// TIA Portal V18 export
FUNCTION_BLOCK "ST10_Flow24_LUnloadingTrans"   // FB1094, GRAPH
VERSION : 0.1
// stored: AcknowledgeErrorsRequired false, AutoNumber false, GraphVersion 6.0, InitialValuesAcquisition false, IsIECCheckEnabled false, LanguageInNetworks LAD, LockOperatingMode false, PermanentILProcessingInMANMode false, SetENOAutomatically false, SkipSteps false, UDAEnableTagReadback false, WithAlarmHandling true
   // inherited from GRAPH_BASE
   VAR
      OFF_SQ_BASE : Bool;
   END_VAR
   VAR_INPUT
      iSysInface : "RCS_SysComInterface_V1";
   END_VAR
   VAR_IN_OUT
      ioPM_Inface : "RCS_PMInterface_V1";
      ioStatus : Int;
   END_VAR
   VAR
      sCtrlMode { S7_SetPoint := 'True'} : "SysFlowCtrlGraph";
      sUpdMES_Data : Bool;   // 更新MES数据
      工件放行中 : Bool;
      前站站号 { ExternalAccessible := 'False'; ExternalVisible := 'False'; ExternalWritable := 'False'} : UInt;
      本站站号 { ExternalAccessible := 'False'; ExternalVisible := 'False'; ExternalWritable := 'False'} : UInt;
      弹窗Temp : Array[1..10] of Int;
      AlarmID : Int;
      TON { S7_SetPoint := 'True'} : Array[0..10] of TON_TIME;
      TOF { S7_SetPoint := 'True'} : Array[0..10] of TOF_TIME;
      sUP { S7_SetPoint := 'True'} : Array[0..10] of Bool;
      更新RFID完成 : Bool;
   END_VAR
   VAR_TEMP
      Tempresult : USInt;
      本站站号乘10 : UInt;
   END_VAR
   // // TON[0] : 托盘流入1托盘到位传感器 / iA-Rotating product Check
   // // TON[1] : 托盘流入1托盘到位传感器
   // // TON[2] : 托盘流入1产品有无传感器
   // // TON[3] : 托盘流入1产品有无传感器
   // // TON[4] : 托盘流入1姿态检测光电2
   // // TON[5] : 托盘流入1姿态检测光电3
   // // TON[0].Q : 托盘流入1托盘到位 / iA-Rotating product Check
   // // TON[1].Q : 托盘流入1托盘无
   // // TON[2].Q : 托盘流入1有产品
   // // TON[3].Q : 托盘流入1无产品
   // // TON[4].Q : 托盘流入1姿态检测光电2
   // // TON[5].Q : 托盘流入1姿态检测光电3
   // // TOF[1] : iA-Rotating product Check
BEGIN
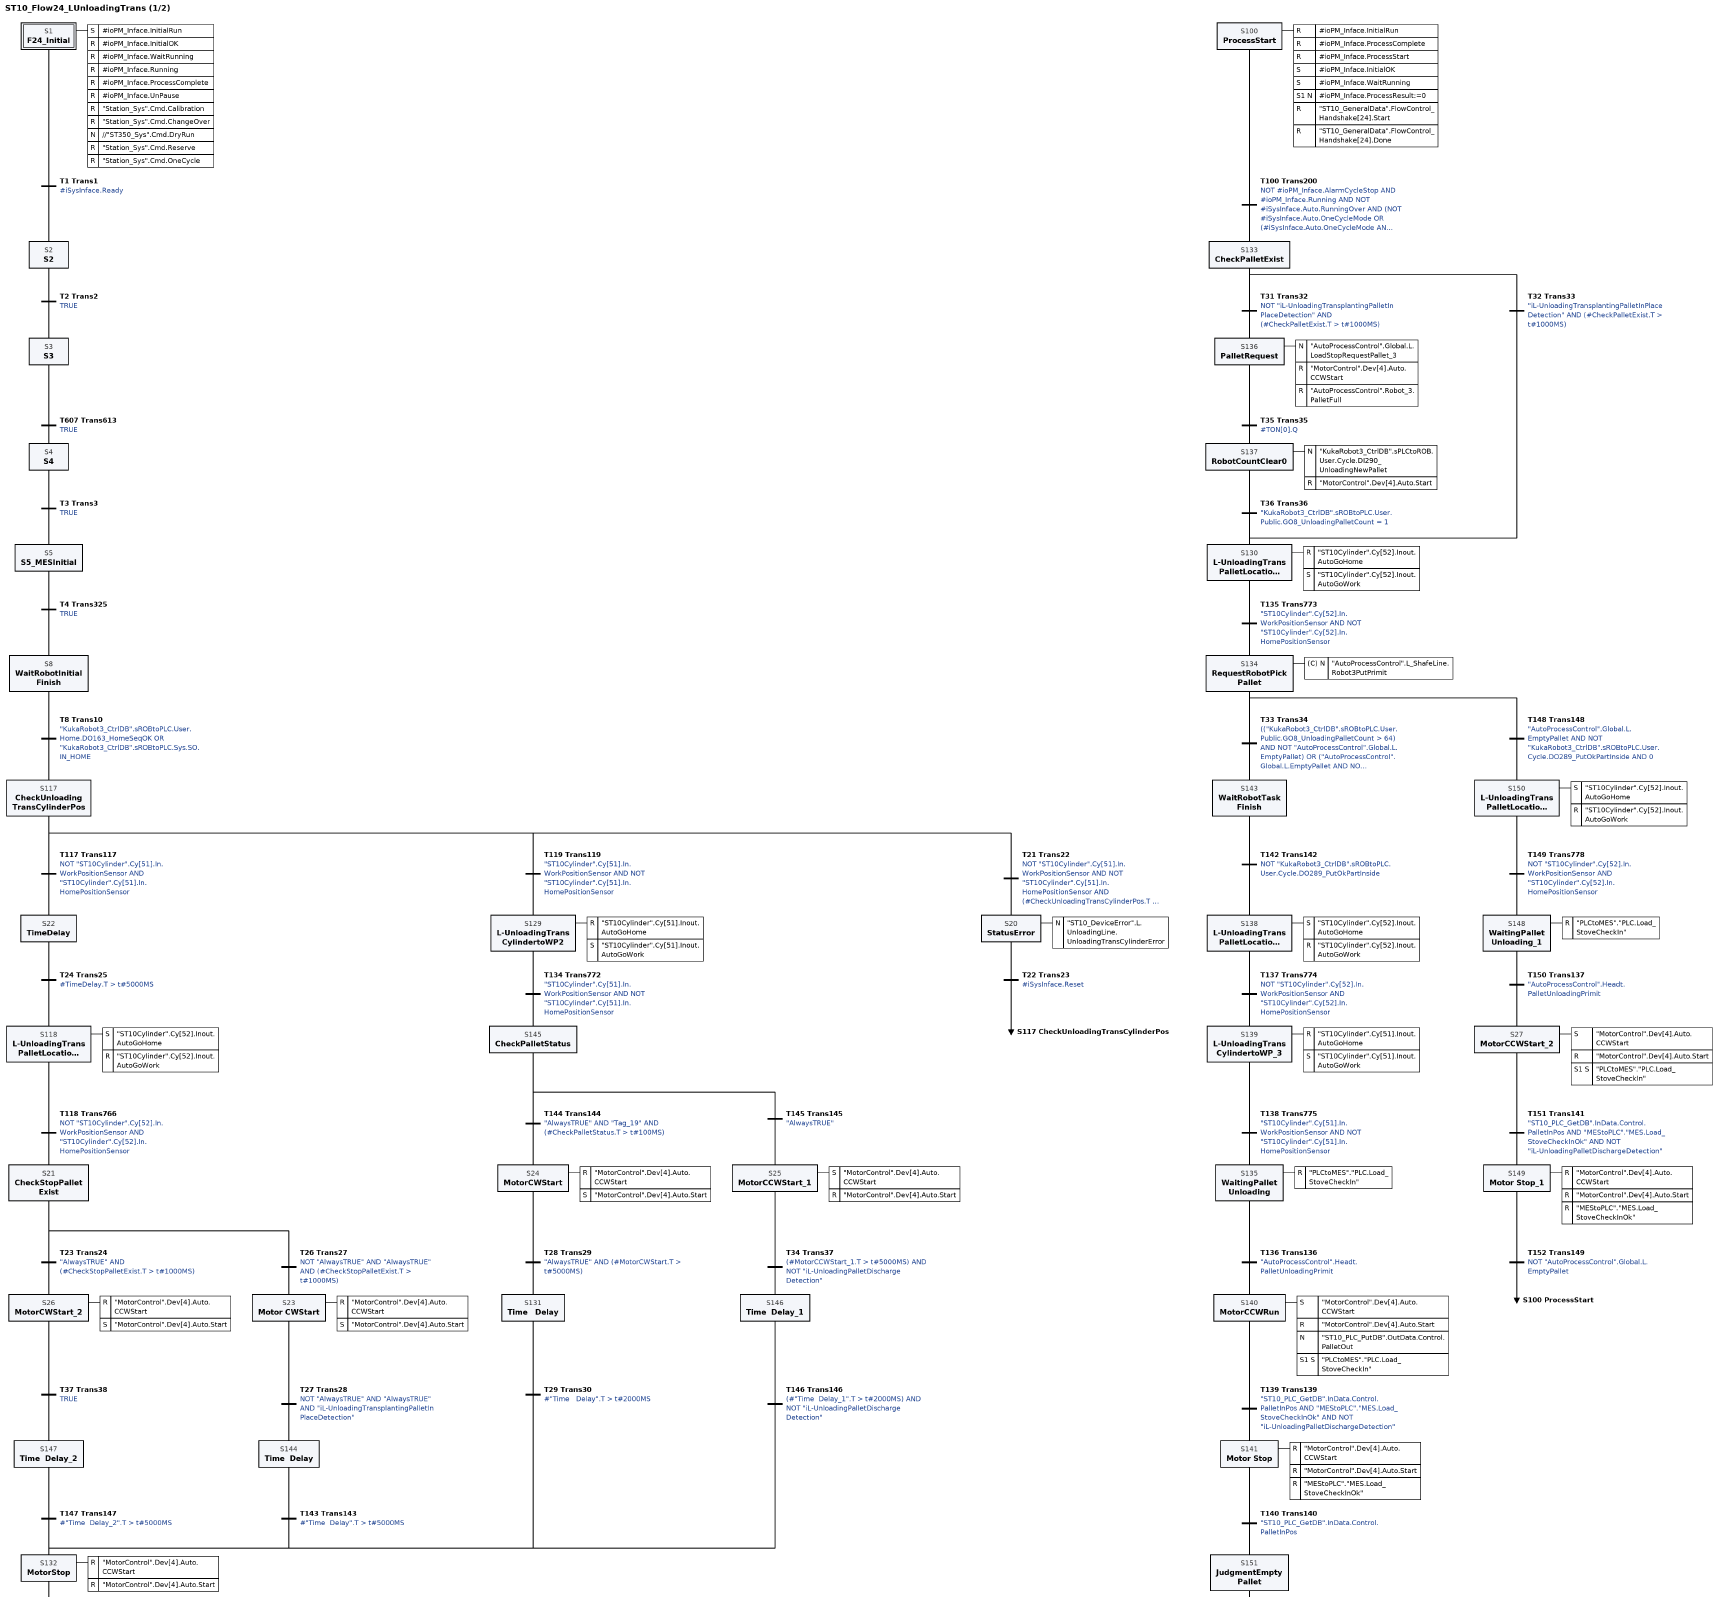
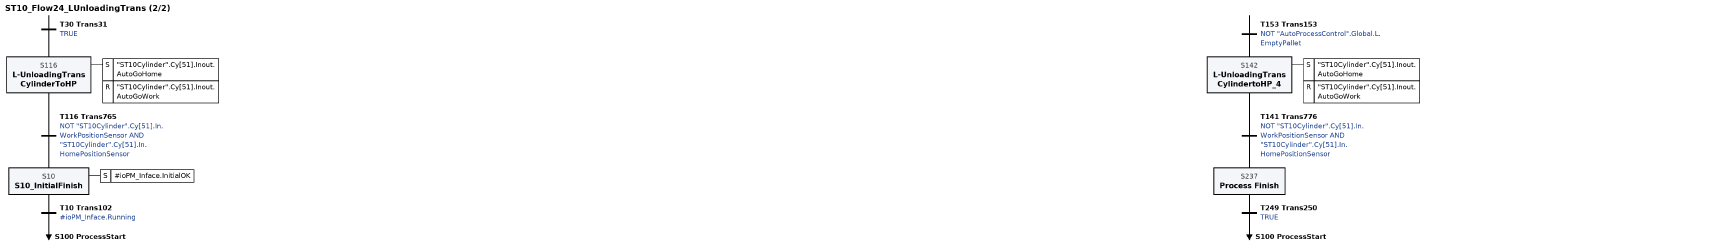
   // permanent pre-instructions
   NETWORK 1
      #TON[10].TON(IN := "AlwaysTRUE" AND "Station_Sys".Alarm.ImmediatelyStop, PT := T#300ms);
      #ioPM_Inface.AlarmImdilyStop := #TON[10].Q;
      #ioPM_Inface.AlarmCycleStop := "AlwaysTRUE" AND "Station_Sys".Alarm.CycleStop;
   NETWORK 2
      IF NOT False THEN
          #sCtrlMode(iSysInface := #iSysInface, ioPM_Inface := #ioPM_Inface, ioGraphCtrl := #RT_DATA.MOP);   // "SysFlowCtrlGraph"
      END_IF;
   NETWORK 3
      #TON[0].TON(IN := "AlwaysTRUE" AND "iL-UnloadingTransplantingPalletInPlaceDetection", PT := t#1000ms);   // 工位11有托盘
      #TOF[1].TOF(IN := "AlwaysTRUE" AND NOT "iL-UnloadingTransplantingPalletInPlaceDetection", PT := T#300ms);   // 工位无托盘
      #TON[2].TON(IN := "AlwaysTRUE", PT := T#300ms);
      #TOF[3].TOF(IN := "AlwaysTRUE", PT := T#300ms);
      #TON[4].TON(IN := "AlwaysTRUE", PT := T#300ms);
      #TOF[5].TOF(IN := "AlwaysTRUE", PT := T#300ms);
   NETWORK 4
      #前站站号 := 345;
      #本站站号 := 350;
   NETWORK 5
      IF "AlwaysTRUE" AND "MEStoPLC"."MES.Load_StoveCheckInOk" THEN
          "PLCtoMES"."PLC.Load_StoveCheckIn" := FALSE;
      END_IF;

   // sequencer 1: S01-S99 初始化 / S01-S99 Initial
   INITIAL_STEP F24_Initial:   // S1, max time T#10S, warning time T#7S
              S    #ioPM_Inface.InitialRun
              R    #ioPM_Inface.InitialOK
              R    #ioPM_Inface.WaitRunning
              R    #ioPM_Inface.Running
              R    #ioPM_Inface.ProcessComplete
              R    #ioPM_Inface.UnPause
              R    "Station_Sys".Cmd.Calibration
              R    "Station_Sys".Cmd.ChangeOver
                   //"ST350_Sys".Cmd.DryRun
              R    "Station_Sys".Cmd.Reserve
              R    "Station_Sys".Cmd.OneCycle
   END_STEP
   TRANSITION Trans1 FROM F24_Initial TO S2   // T1
      := #iSysInface.Ready;
   END_TRANSITION
   STEP S2:   // S2, max time T#10S, warning time T#7S
   END_STEP
   TRANSITION Trans2 FROM S2 TO S3   // T2
      := TRUE;
   END_TRANSITION
   STEP S4:   // S4, max time T#10S, warning time T#7S
   END_STEP
   TRANSITION Trans3 FROM S4 TO S5_MESInitial   // T3
      := TRUE;
   END_TRANSITION
   STEP S5_MESInitial:   // S5, max time T#10S, warning time T#7S
   END_STEP
   TRANSITION Trans325 FROM S5_MESInitial TO WaitRobotInitialFinish   // T4
      := TRUE;
   END_TRANSITION
   STEP S10_InitialFinish:   // S10, max time T#10S, warning time T#7S
              S    #ioPM_Inface.InitialOK
   END_STEP
   TRANSITION Trans102 FROM S10_InitialFinish TO ProcessStart   // T10, jump
      := #ioPM_Inface.Running;
   END_TRANSITION
   STEP S3:   // S3, max time T#10S, warning time T#7S
   END_STEP
   TRANSITION Trans613 FROM S3 TO S4   // T607
      := TRUE;
   END_TRANSITION
   STEP WaitRobotInitialFinish:   // S8, max time T#10S, warning time T#7S
   END_STEP
   TRANSITION Trans10 FROM WaitRobotInitialFinish TO CheckUnloadingTransCylinderPos   // T8
      := "KukaRobot3_CtrlDB".sROBtoPLC.User.Home.DO163_HomeSeqOK OR "KukaRobot3_CtrlDB".sROBtoPLC.Sys.SO.IN_HOME;
   END_TRANSITION
   STEP "Time   Delay":   // S131, max time T#10S, warning time T#7S
   END_STEP
   TRANSITION Trans30 FROM "Time   Delay" TO MotorStop   // T29
      := #"Time   Delay".T > t#2000MS;
   END_TRANSITION
   STEP CheckUnloadingTransCylinderPos:   // S117, max time T#10S, warning time T#7S
   END_STEP
   TRANSITION Trans117 FROM CheckUnloadingTransCylinderPos TO TimeDelay   // T117
      := NOT "ST10Cylinder".Cy[51].In.WorkPositionSensor AND "ST10Cylinder".Cy[51].In.HomePositionSensor;
   END_TRANSITION
   TRANSITION Trans119 FROM CheckUnloadingTransCylinderPos TO "L-UnloadingTransCylindertoWP2"   // T119
      := "ST10Cylinder".Cy[51].In.WorkPositionSensor AND NOT "ST10Cylinder".Cy[51].In.HomePositionSensor;
   END_TRANSITION
   TRANSITION Trans22 FROM CheckUnloadingTransCylinderPos TO StatusError   // T21
      := NOT "ST10Cylinder".Cy[51].In.WorkPositionSensor AND NOT "ST10Cylinder".Cy[51].In.HomePositionSensor AND (#CheckUnloadingTransCylinderPos.T > t#2000MS);
   END_TRANSITION
   STEP "L-UnloadingTransCylinderToHP":   // S116, max time T#10S, warning time T#7S
              S    "ST10Cylinder".Cy[51].Inout.AutoGoHome
              R    "ST10Cylinder".Cy[51].Inout.AutoGoWork
   END_STEP
   TRANSITION Trans765 FROM "L-UnloadingTransCylinderToHP" TO S10_InitialFinish   // T116
      := NOT "ST10Cylinder".Cy[51].In.WorkPositionSensor AND "ST10Cylinder".Cy[51].In.HomePositionSensor;
   END_TRANSITION
   STEP StatusError:   // S20, max time T#10S, warning time T#7S
              N    "ST10_DeviceError".L.UnloadingLine.UnloadingTransCylinderError
   END_STEP
   TRANSITION Trans23 FROM StatusError TO CheckUnloadingTransCylinderPos   // T22, jump
      := #iSysInface.Reset;
   END_TRANSITION
   STEP CheckStopPalletExist:   // S21, max time T#10S, warning time T#7S
   END_STEP
   TRANSITION Trans24 FROM CheckStopPalletExist TO MotorCWStart_2   // T23
      := "AlwaysTRUE" AND (#CheckStopPalletExist.T > t#1000MS);
   END_TRANSITION
   TRANSITION Trans27 FROM CheckStopPalletExist TO "Motor CWStart"   // T26
      := NOT "AlwaysTRUE" AND "AlwaysTRUE" AND (#CheckStopPalletExist.T > t#1000MS);
   END_TRANSITION
   STEP TimeDelay:   // S22, max time T#10S, warning time T#7S
   END_STEP
   TRANSITION Trans25 FROM TimeDelay TO "L-UnloadingTransPalletLocationCylinderHP_2"   // T24
      := #TimeDelay.T > t#5000MS;
   END_TRANSITION
   STEP "Motor CWStart":   // S23, max time T#10S, warning time T#7S
              R    "MotorControl".Dev[4].Auto.CCWStart
              S    "MotorControl".Dev[4].Auto.Start
   END_STEP
   TRANSITION Trans28 FROM "Motor CWStart" TO "Time  Delay"   // T27
      := NOT "AlwaysTRUE" AND "AlwaysTRUE" AND "iL-UnloadingTransplantingPalletInPlaceDetection";
   END_TRANSITION
   STEP MotorCWStart:   // S24, max time T#10S, warning time T#7S
              R    "MotorControl".Dev[4].Auto.CCWStart
              S    "MotorControl".Dev[4].Auto.Start
   END_STEP
   TRANSITION Trans29 FROM MotorCWStart TO "Time   Delay"   // T28
      := "AlwaysTRUE" AND (#MotorCWStart.T > t#5000MS);
   END_TRANSITION
   STEP "L-UnloadingTransCylindertoWP2":   // S129, max time T#10S, warning time T#7S
              R    "ST10Cylinder".Cy[51].Inout.AutoGoHome
              S    "ST10Cylinder".Cy[51].Inout.AutoGoWork
   END_STEP
   TRANSITION Trans772 FROM "L-UnloadingTransCylindertoWP2" TO CheckPalletStatus   // T134
      := "ST10Cylinder".Cy[51].In.WorkPositionSensor AND NOT "ST10Cylinder".Cy[51].In.HomePositionSensor;
   END_TRANSITION
   STEP MotorStop:   // S132, max time T#10S, warning time T#7S
              R    "MotorControl".Dev[4].Auto.CCWStart
              R    "MotorControl".Dev[4].Auto.Start
   END_STEP
   TRANSITION Trans31 FROM MotorStop TO "L-UnloadingTransCylinderToHP"   // T30
      := TRUE;
   END_TRANSITION
   STEP "L-UnloadingTransPalletLocationCylinderHP_2":   // S118, max time T#10S, warning time T#7S
              S    "ST10Cylinder".Cy[52].Inout.AutoGoHome
              R    "ST10Cylinder".Cy[52].Inout.AutoGoWork
   END_STEP
   TRANSITION Trans766 FROM "L-UnloadingTransPalletLocationCylinderHP_2" TO CheckStopPalletExist   // T118
      := NOT "ST10Cylinder".Cy[52].In.WorkPositionSensor AND "ST10Cylinder".Cy[52].In.HomePositionSensor;
   END_TRANSITION
   STEP "Time  Delay":   // S144, max time T#10S, warning time T#7S
   END_STEP
   TRANSITION Trans143 FROM "Time  Delay" TO MotorStop   // T143
      := #"Time  Delay".T > t#5000MS;
   END_TRANSITION
   STEP CheckPalletStatus:   // S145, max time T#10S, warning time T#7S
   END_STEP
   TRANSITION Trans144 FROM CheckPalletStatus TO MotorCWStart   // T144
      := "AlwaysTRUE" AND "Tag_19" AND (#CheckPalletStatus.T > t#100MS);
   END_TRANSITION
   TRANSITION Trans145 FROM CheckPalletStatus TO MotorCCWStart_1   // T145
      := "AlwaysTRUE";
   END_TRANSITION
   STEP MotorCCWStart_1:   // S25, max time T#10S, warning time T#7S
              S    "MotorControl".Dev[4].Auto.CCWStart
              R    "MotorControl".Dev[4].Auto.Start
   END_STEP
   TRANSITION Trans37 FROM MotorCCWStart_1 TO "Time  Delay_1"   // T34
      := (#MotorCCWStart_1.T > t#5000MS) AND NOT "iL-UnloadingPalletDischargeDetection";
   END_TRANSITION
   STEP "Time  Delay_1":   // S146, max time T#10S, warning time T#7S
   END_STEP
   TRANSITION Trans146 FROM "Time  Delay_1" TO MotorStop   // T146
      := (#"Time  Delay_1".T > t#2000MS) AND NOT "iL-UnloadingPalletDischargeDetection";
   END_TRANSITION
   STEP MotorCWStart_2:   // S26, max time T#10S, warning time T#7S
              R    "MotorControl".Dev[4].Auto.CCWStart
              S    "MotorControl".Dev[4].Auto.Start
   END_STEP
   TRANSITION Trans38 FROM MotorCWStart_2 TO "Time  Delay_2"   // T37
      := TRUE;
   END_TRANSITION
   STEP "Time  Delay_2":   // S147, max time T#10S, warning time T#7S
   END_STEP
   TRANSITION Trans147 FROM "Time  Delay_2" TO MotorStop   // T147
      := #"Time  Delay_2".T > t#5000MS;
   END_TRANSITION

   // sequencer 2: S100-S199 等待到位 / S100-S199 CheckPalletStatus
   STEP ProcessStart:   // S100, max time T#10S, warning time T#7S
      // 自动等待开始运行
              R    #ioPM_Inface.InitialRun
              R    #ioPM_Inface.ProcessComplete
              R    #ioPM_Inface.ProcessStart
              S    #ioPM_Inface.InitialOK
              S    #ioPM_Inface.WaitRunning
          S1  N    #ioPM_Inface.ProcessResult:=0
              R    "ST10_GeneralData".FlowControl_Handshake[24].Start
              R    "ST10_GeneralData".FlowControl_Handshake[24].Done
   END_STEP
   TRANSITION Trans200 FROM ProcessStart TO CheckPalletExist   // T100
      := NOT #ioPM_Inface.AlarmCycleStop AND #ioPM_Inface.Running AND NOT #iSysInface.Auto.RunningOver AND (NOT #iSysInface.Auto.OneCycleMode OR (#iSysInface.Auto.OneCycleMode AND #ioPM_Inface.TriggerOneCycle));
   END_TRANSITION
   STEP "Process Finish":   // S237, max time T#10S, warning time T#7S
   END_STEP
   TRANSITION Trans250 FROM "Process Finish" TO ProcessStart   // T249, jump
      := TRUE;
   END_TRANSITION
   STEP PalletRequest:   // S136, max time T#10S, warning time T#7S
              N    "AutoProcessControl".Global.L.LoadStopRequestPallet_3
              R    "MotorControl".Dev[4].Auto.CCWStart
              R    "AutoProcessControl".Robot_3.PalletFull
   END_STEP
   TRANSITION Trans35 FROM PalletRequest TO RobotCountClear0   // T35
      := #TON[0].Q;
   END_TRANSITION
   STEP WaitingPalletUnloading:   // S135, max time T#10S, warning time T#7S
              R    "PLCtoMES"."PLC.Load_StoveCheckIn"
   END_STEP
   TRANSITION Trans136 FROM WaitingPalletUnloading TO MotorCCWRun   // T136
      := "AutoProcessControl".Headt.PalletUnloadingPrimit;
   END_TRANSITION
   STEP RequestRobotPickPallet:   // S134, max time T#10S, warning time T#7S
      interlock C := NOT "AutoProcessControl".Robot_3.PalletFull AND NOT "AutoProcessControl".Global.L.EmptyPallet;
      (C)     N    "AutoProcessControl".L_ShafeLine.Robot3PutPrimit
   END_STEP
   TRANSITION Trans34 FROM RequestRobotPickPallet TO WaitRobotTaskFinish   // T33
      := (("KukaRobot3_CtrlDB".sROBtoPLC.User.Public.GO8_UnloadingPalletCount > 64) AND NOT "AutoProcessControl".Global.L.EmptyPallet) OR ("AutoProcessControl".Global.L.EmptyPallet AND NOT "KukaRobot3_CtrlDB".sROBtoPLC.User.Cycle.DO289_PutOkPartInside) OR ("AutoProcessControl".Robot_3.PalletFull AND "iL-UnloadingTransplantingPalletInPlaceDetection" AND NOT "KukaRobot3_CtrlDB".sROBtoPLC.User.Cycle.DO289_PutOkPartInside AND (#RequestRobotPickPallet.T > t#5000MS) AND NOT "AutoProcessControl".Global.L.EmptyPallet);
   END_TRANSITION
   TRANSITION Trans148 FROM RequestRobotPickPallet TO "L-UnloadingTransPalletLocationCylinderTo HP_1"   // T148
      := "AutoProcessControl".Global.L.EmptyPallet AND NOT "KukaRobot3_CtrlDB".sROBtoPLC.User.Cycle.DO289_PutOkPartInside AND 0;
   END_TRANSITION
   STEP RobotCountClear0:   // S137, max time T#10S, warning time T#7S
              N    "KukaRobot3_CtrlDB".sPLCtoROB.User.Cycle.DI290_UnloadingNewPallet
              R    "MotorControl".Dev[4].Auto.Start
   END_STEP
   TRANSITION Trans36 FROM RobotCountClear0 TO "L-UnloadingTransPalletLocationCylinder ToWP"   // T36
      := "KukaRobot3_CtrlDB".sROBtoPLC.User.Public.GO8_UnloadingPalletCount = 1;
   END_TRANSITION
   STEP CheckPalletExist:   // S133, max time T#10S, warning time T#7S
   END_STEP
   TRANSITION Trans32 FROM CheckPalletExist TO PalletRequest   // T31
      := NOT "iL-UnloadingTransplantingPalletInPlaceDetection" AND (#CheckPalletExist.T > t#1000MS);
   END_TRANSITION
   TRANSITION Trans33 FROM CheckPalletExist TO "L-UnloadingTransPalletLocationCylinder ToWP"   // T32
      := "iL-UnloadingTransplantingPalletInPlaceDetection" AND (#CheckPalletExist.T > t#1000MS);
   END_TRANSITION
   STEP "L-UnloadingTransPalletLocationCylinder ToWP":   // S130, max time T#10S, warning time T#7S
              R    "ST10Cylinder".Cy[52].Inout.AutoGoHome
              S    "ST10Cylinder".Cy[52].Inout.AutoGoWork
   END_STEP
   TRANSITION Trans773 FROM "L-UnloadingTransPalletLocationCylinder ToWP" TO RequestRobotPickPallet   // T135
      := "ST10Cylinder".Cy[52].In.WorkPositionSensor AND NOT "ST10Cylinder".Cy[52].In.HomePositionSensor;
   END_TRANSITION
   STEP "L-UnloadingTransPalletLocationCylinderTo HP":   // S138, max time T#10S, warning time T#7S
              S    "ST10Cylinder".Cy[52].Inout.AutoGoHome
              R    "ST10Cylinder".Cy[52].Inout.AutoGoWork
   END_STEP
   TRANSITION Trans774 FROM "L-UnloadingTransPalletLocationCylinderTo HP" TO "L-UnloadingTransCylindertoWP_3"   // T137
      := NOT "ST10Cylinder".Cy[52].In.WorkPositionSensor AND "ST10Cylinder".Cy[52].In.HomePositionSensor;
   END_TRANSITION
   STEP "L-UnloadingTransCylindertoWP_3":   // S139, max time T#10S, warning time T#7S
              R    "ST10Cylinder".Cy[51].Inout.AutoGoHome
              S    "ST10Cylinder".Cy[51].Inout.AutoGoWork
   END_STEP
   TRANSITION Trans775 FROM "L-UnloadingTransCylindertoWP_3" TO WaitingPalletUnloading   // T138
      := "ST10Cylinder".Cy[51].In.WorkPositionSensor AND NOT "ST10Cylinder".Cy[51].In.HomePositionSensor;
   END_TRANSITION
   STEP MotorCCWRun:   // S140, max time T#10S, warning time T#7S
              S    "MotorControl".Dev[4].Auto.CCWStart
              R    "MotorControl".Dev[4].Auto.Start
              N    "ST10_PLC_PutDB".OutData.Control.PalletOut
          S1  S    "PLCtoMES"."PLC.Load_StoveCheckIn"
   END_STEP
   TRANSITION Trans139 FROM MotorCCWRun TO "Motor Stop"   // T139
      := "ST10_PLC_GetDB".InData.Control.PalletInPos AND "MEStoPLC"."MES.Load_StoveCheckInOk" AND NOT "iL-UnloadingPalletDischargeDetection";
   END_TRANSITION
   STEP "Motor Stop":   // S141, max time T#10S, warning time T#7S
              R    "MotorControl".Dev[4].Auto.CCWStart
              R    "MotorControl".Dev[4].Auto.Start
              R    "MEStoPLC"."MES.Load_StoveCheckInOk"
   END_STEP
   TRANSITION Trans140 FROM "Motor Stop" TO JudgmentEmptyPallet   // T140
      := "ST10_PLC_GetDB".InData.Control.PalletInPos;
   END_TRANSITION
   STEP "L-UnloadingTransCylindertoHP_4":   // S142, max time T#10S, warning time T#7S
              S    "ST10Cylinder".Cy[51].Inout.AutoGoHome
              R    "ST10Cylinder".Cy[51].Inout.AutoGoWork
   END_STEP
   TRANSITION Trans776 FROM "L-UnloadingTransCylindertoHP_4" TO "Process Finish"   // T141
      := NOT "ST10Cylinder".Cy[51].In.WorkPositionSensor AND "ST10Cylinder".Cy[51].In.HomePositionSensor;
   END_TRANSITION
   STEP WaitRobotTaskFinish:   // S143, max time T#10S, warning time T#7S
   END_STEP
   TRANSITION Trans142 FROM WaitRobotTaskFinish TO "L-UnloadingTransPalletLocationCylinderTo HP"   // T142
      := NOT "KukaRobot3_CtrlDB".sROBtoPLC.User.Cycle.DO289_PutOkPartInside;
   END_TRANSITION
   STEP "L-UnloadingTransPalletLocationCylinderTo HP_1":   // S150, max time T#10S, warning time T#7S
              S    "ST10Cylinder".Cy[52].Inout.AutoGoHome
              R    "ST10Cylinder".Cy[52].Inout.AutoGoWork
   END_STEP
   TRANSITION Trans778 FROM "L-UnloadingTransPalletLocationCylinderTo HP_1" TO WaitingPalletUnloading_1   // T149
      := NOT "ST10Cylinder".Cy[52].In.WorkPositionSensor AND "ST10Cylinder".Cy[52].In.HomePositionSensor;
   END_TRANSITION
   STEP MotorCCWStart_2:   // S27, max time T#10S, warning time T#7S
              S    "MotorControl".Dev[4].Auto.CCWStart
              R    "MotorControl".Dev[4].Auto.Start
          S1  S    "PLCtoMES"."PLC.Load_StoveCheckIn"
   END_STEP
   TRANSITION Trans141 FROM MotorCCWStart_2 TO "Motor Stop_1"   // T151
      := "ST10_PLC_GetDB".InData.Control.PalletInPos AND "MEStoPLC"."MES.Load_StoveCheckInOk" AND NOT "iL-UnloadingPalletDischargeDetection";
   END_TRANSITION
   STEP WaitingPalletUnloading_1:   // S148, max time T#10S, warning time T#7S
              R    "PLCtoMES"."PLC.Load_StoveCheckIn"
   END_STEP
   TRANSITION Trans137 FROM WaitingPalletUnloading_1 TO MotorCCWStart_2   // T150
      := "AutoProcessControl".Headt.PalletUnloadingPrimit;
   END_TRANSITION
   STEP "Motor Stop_1":   // S149, max time T#10S, warning time T#7S
              R    "MotorControl".Dev[4].Auto.CCWStart
              R    "MotorControl".Dev[4].Auto.Start
              R    "MEStoPLC"."MES.Load_StoveCheckInOk"
   END_STEP
   TRANSITION Trans149 FROM "Motor Stop_1" TO ProcessStart   // T152, jump
      := NOT "AutoProcessControl".Global.L.EmptyPallet;
   END_TRANSITION
   STEP JudgmentEmptyPallet:   // S151, max time T#10S, warning time T#7S
   END_STEP
   TRANSITION Trans153 FROM JudgmentEmptyPallet TO "L-UnloadingTransCylindertoHP_4"   // T153
      := NOT "AutoProcessControl".Global.L.EmptyPallet;
   END_TRANSITION

   // permanent post-instructions
   NETWORK 1
      #ioPM_Inface.StepNum := #RT_DATA.S_DISPLAY;
   NETWORK 2
      IF #iSysInface.Reset THEN #AlarmID := 0; END_IF;
   NETWORK 3
      #TON[10].TON(IN := #工件放行中, PT := T#0.5S);
      IF #TON[10].Q THEN #工件放行中 := FALSE; END_IF;
END_FUNCTION_BLOCK
